(*
SPDX-FileCopyrightText: © 2026 Oleksandr Tiutyk <trofimich@gmail.com>
SPDX-License-Identifier: MIT
License: https://opensource.org/license/mit
*)

INTERFACE IDataMemberTypeNotSupportedException EXTENDS IGeneralException

METHOD Throw
VAR_INPUT
	sourceNamespaceName : STRING;
	sourceClassName : STRING;
	sourcePOUName : STRING;
	sourcePosition : STRING;
	dataMemberName : STRING;
	dataMemberTypeName : STRING;
END_VAR
END_METHOD

END_INTERFACE

(* stored: Version 1.1.0.1
   Itf IDataMemberTypeNotSupportedException: Id {11c08bf0-c6ce-49fe-8b89-9f8f5e6c5095}
   Method Throw: Id {d75368a2-4715-4ba7-89d0-da1934b67c1e} *)
